// TIA Portal V20 export
DATA_BLOCK "DB_Alarm"   // DB13
// stored: Access Published, MemoryReserve 100, Namespace LineA1
   VAR
      "word" : Struct
         Line : Struct
            A1 : Struct
               Conveyor : Array[_.minA1.._.maxA1] of Word;
            END_STRUCT;
         END_STRUCT;
      END_STRUCT;
   END_VAR
BEGIN
END_DATA_BLOCK
